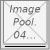
VISUALIZATION F_MainMenu_04  // 50x50
VAR_IN_OUT
	stMenuButton	: ST_HMIEButton_HMI;
END_VAR
    Image (3,0 44x44), invisible if: not stMenuButton.bVisible, image: ImagePool.04_ChangeMode
        OnMouseDown: execute { stMenuButton.bPushed := TRUE; }
    Line (5,46) (45,46), invisible if: not stMenuButton.bVisible or not stMenuButton.bActive, input disabled if: not stMenuButton.bEnable
END_VISUALIZATION

(* stored: Version 1.1.0.1
   Visu F_MainMenu_04: Id {c81f1ef8-fe0d-0c10-2291-8e9c76e48f27} *)
